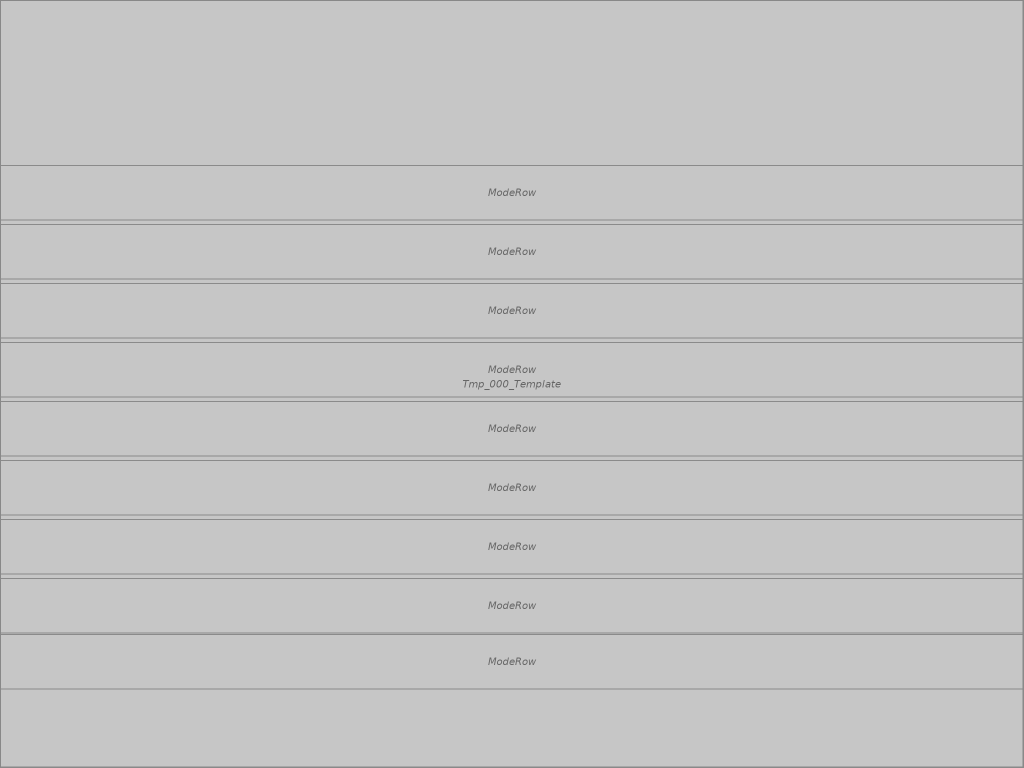
VISUALIZATION Mod_002_ModeScreenRows  // 1024x768
    Frame (0,0 1024x768)
        shows Tmp_000_Template(header := gHMIData.hmiHeader)
    Frame (0,165 1024x55)
        shows ModeRow(MotionRowInstanceSingle := gModeAlternate.gModeRows.gMotionRow1, MotionRowButtonsSingle := gModeAlternate.gModeButtons.gMotionRow1btn)
    Frame (0,224 1024x55)
        shows ModeRow(MotionRowInstanceSingle := gModeAlternate.gModeRows.gMotionRow2, MotionRowButtonsSingle := gModeAlternate.gModeButtons.gMotionRow2btn)
    Frame (0,283 1024x55)
        shows ModeRow(MotionRowInstanceSingle := gModeAlternate.gModeRows.gMotionRow3, MotionRowButtonsSingle := gModeAlternate.gModeButtons.gMotionRow3btn)
    Frame (0,342 1024x55)
        shows ModeRow(MotionRowInstanceSingle := gModeAlternate.gModeRows.gMotionRow4, MotionRowButtonsSingle := gModeAlternate.gModeButtons.gMotionRow4btn)
    Frame (0,401 1024x55)
        shows ModeRow(MotionRowInstanceSingle := gModeAlternate.gModeRows.gMotionRow5, MotionRowButtonsSingle := gModeAlternate.gModeButtons.gMotionRow5btn)
    Frame (0,460 1024x55)
        shows ModeRow(MotionRowInstanceSingle := gModeAlternate.gModeRows.gMotionRow6, MotionRowButtonsSingle := gModeAlternate.gModeButtons.gMotionRow6btn)
    Frame (0,519 1024x55)
        shows ModeRow(MotionRowInstanceSingle := gModeAlternate.gModeRows.gMotionRow7, MotionRowButtonsSingle := gModeAlternate.gModeButtons.gMotionRow7btn)
    Frame (0,578 1024x55)
        shows ModeRow(MotionRowInstanceSingle := gModeAlternate.gModeRows.gMotionRow8, MotionRowButtonsSingle := gModeAlternate.gModeButtons.gMotionRow8btn)
    Frame (0,634 1024x55)
        shows ModeRow(MotionRowInstanceSingle := gModeAlternate.gModeRows.gMotionRow9, MotionRowButtonsSingle := gModeAlternate.gModeButtons.gMotionRow9btn)
END_VISUALIZATION

(* stored: Version 1.1.0.1, ProductVersion 3.1.4024.12
   Visu Mod_002_ModeScreenRows: Id {8382fd68-021f-4212-b7a3-3e83aa5706fa} *)
